// TIA Portal V19 export
TYPE "LEXCHANGETRAY_typeNgConveyor_toHandlingXyzDeliver"
// stored: Access Published
   STRUCT
      feedback : "LEXCHANGETRAY_typeNgConveyorEm_toHandlingXyzFeedback";
      req : "LEXCHANGETRAY_typeNgConveyorEm_toHandlingXyzReq";
   END_STRUCT;
END_TYPE
